{library PUBLIC}
(*
Sequence for a specific device during send or receive on level 2.
This can be used for debug but is only visible inside a block.
 *)
TYPE DEVICE_SEQUENCE :
(
	DEVICE_SEQUENCE_NOP:=0,							(* No operation - free *)
	DEVICE_SEQUENCE_INIT,							(* Init of block *)
	DEVICE_SEQUENCE_WAIT_FOR_DEVICE_READY,			(* Prepare for wait and set busy to true *)
	DEVICE_SEQUENCE_WAIT_FOR_STROBE_LOW,			(* Wait until target device strobe and data are 0 *)
	DEVICE_SEQUENCE_PREPARE_SEND_RECEIVE,
	DEVICE_SEQUENCE_STROBE_HIGH,
	DEVICE_SEQUENCE_SEND_RECEIVE,					(* Transfer or read data *)
	DEVICE_SEQUENCE_ACK,
	DEVICE_SEQUENCE_WAIT_FOR_ANSWER,
	DEVICE_SEQUENCE_SET_LOW,						(* Data and strobe to 0 *)
	DEVICE_SEQUENCE_READY,							(* End of sequence will wait in this step until En=false *)

	DEVICE_SEQUENCE_TIME_OUT:=-1,					(* Tinme out during send or receive *)
	DEVICE_SEQUENCE_CANCEL:=-2,						(* An ongoing operation was canceld *)
	DEVICE_SEQUENCE_ERROR:=-3						(* An error during send/receive *)
);
END_TYPE
//  DEVICE_SEQUENCE_TIME_OUT = '-1'
//  DEVICE_SEQUENCE_CANCEL = '-2'
//  DEVICE_SEQUENCE_ERROR = '-3'

(* stored: Version 1.1.0.1, ProductVersion 3.1.4024.2
   EnumerationTextList DEVICE_SEQUENCE: Id {3679e7c3-6e6a-47d6-8bcc-f60ab5402f9c} *)
